(*
A broadcastable wrapper for a `DWORD` value. 
*)
INTERFACE I_DwordArg EXTENDS I_Arg

(*
Reads the internal value.
*)
PROPERTY Get : DWORD
GET
END_GET
END_PROPERTY

(*
Returns TRUE if the value is mutable.
*)
PROPERTY IsMut : BOOL
GET
END_GET
END_PROPERTY

(*
Modifies the internal value.  
Returns:
- `Ok` - Upon successful modification.
- `Error` - If mutability is disabled.
*)
METHOD Set : Result
VAR_INPUT
	newVal		: DWORD;
END_VAR
END_METHOD

END_INTERFACE

(* stored: Version 1.1.0.1
   Itf I_DwordArg: Id {94d22b80-e454-4af8-9287-79e03c1786c6}
   Property Get: Id {48310225-1096-4de5-8eab-a38070bbfe2d}
   Get Get: Id {dfe94c58-a283-47cf-b259-8eeb403757b7}
   Property IsMut: Id {3c72062c-3ed0-484f-900e-47f0e01c24cb}
   Get Get: Id {4ea02e19-9b9c-4226-bb7d-c44527921603}
   Method Set: Id {c9a1a77a-4bbb-474d-90ef-783a07cdd625} *)
